(* PLC project v0.6.04_CycleSemiAuto.project, CODESYS CODESYS V3.5 SP19 Patch 1 *)
(* stored: creationDateTime 2026-08-11T14:02:33.650710, modificationDateTime 2026-08-11T14:02:33.650710 *)

(* ═══════════════════════════════════════════════════════════════ 🔧 ST_TranslationCfg — Configurations et paramètres réglables pour Translation M3 ─────────────────────────────────────────────────────────────── 🎨 Destiné au paramétrage depuis l'IHM (RETAIN) — même patron que ST_WinchCfg. 📄 2026-08-06 : créé suite constat terrain — Translation n'avait pas de slot Cfg (contrairement à ST_WinchHMI), les 3 vitesses de ralentissement d'approche n'étaient donc réglables qu'en dur dans GVL_PERSISTENT (recompilation requise). ═══════════════════════════════════════════════════════════════ *)
TYPE ST_TranslationCfg : STRUCT
  CfgApproachSpeedTremie_Hz : REAL := 10;  (* 🐢 Vitesse réduite d'approche Trémie (Hz), déclenchée par capteur PV, Direction=1 *)
  CfgApproachSpeedMaintenance_Hz : REAL := 10;  (* 🐢 Vitesse réduite d'approche Maintenance (Hz), déclenchée par capteur P1, Direction=-1 *)
  CfgApproachSpeedP1_Hz : REAL := 10;  (* 🐢 Vitesse réduite d'approche P1 (Hz), déclenchée par capteur P2, Direction=-1 *)
  Initialized : BOOL := FALSE;  (* 🐛 Flag restauration boot (défaut FALSE non ambigu) — même patron que ST_WinchCfg 🚦 TRUE = config restaurée depuis GVL_PERSISTENT ce boot *)
END_STRUCT;
END_TYPE

(* ═══════════════════════════════════════════════════════════════ 🌉 FB_CfgPersistBridge_TranslationCfg — Pont persistance générique pour ST_TranslationCfg ─────────────────────────────────────────────────────────────── 🎯 Instance unique : TranslationM3.Cfg (un seul axe M3, contrairement à M1/M2). Restaure Persist → Hmi au boot si nécessaire, puis sauvegarde Hmi → Persist. ═══════════════════════════════════════════════════════════════ *)
FUNCTION_BLOCK FB_CfgPersistBridge_TranslationCfg
  VAR_OUTPUT
    JustRestored : BOOL;  (* 🔔 TRUE pendant le scan de restauration *)
  END_VAR
  VAR_IN_OUT
    Hmi : ST_TranslationCfg;  (* 🖥️ Struct exposé à l'IHM *)
    Persist : ST_TranslationCfg;  (* 💾 Mémoire PERSISTENT *)
  END_VAR

            

JustRestored := FALSE;
IF NOT Hmi.Initialized THEN
    Hmi := Persist;
    Hmi.Initialized := TRUE;
    JustRestored := TRUE;
ELSE
    Persist := Hmi;
END_IF;

          
END_FUNCTION_BLOCK
